// TIA Portal V17 export
// export: Created 2022-07-28T18:02:48.2971435Z, ExportSetting None, DisplayName Totally Integrated Automation Portal, DisplayVersion V17, DisplayName TIA Portal Openness, DisplayVersion V17, DisplayName TIA Portal Teamcenter Gateway, DisplayVersion V17, DisplayName TIA Portal Version Control Interface, DisplayVersion V17, DisplayName TIA Portal Test Suite Advanced, DisplayVersion V17, DisplayName SINAMICS Startdrive Advanced, DisplayVersion V17, DisplayName SINAMICS DCC, DisplayVersion V17, DisplayName SINAMICS Startdrive G130, G150, S120, S150, SINAMICS MV, S210, DisplayVersion V17, DisplayName SINAMICS Startdrive G110M, G120, G120C, G120D, G120P, G115D, DisplayVersion V17, DisplayName STEP 7 Professional, DisplayVersion V17, DisplayName SIMATIC Energy Suite, DisplayVersion V17, DisplayName STEP 7 CFC, DisplayVersion V17, DisplayName STEP 7 Safety, DisplayVersion V17, DisplayName WinCC Advanced / Unified PC, DisplayVersion V17, DisplayName SIMATIC Visualization Architect, DisplayVersion V17
FUNCTION "PID_FC" : Void   // FC21, SCL
{ S7_Optimized_Access := 'TRUE' }
// stored: AutoNumber false, SetENOAutomatically false
   VAR_TEMP
      t_SupplyRelease : Bool;   // 1 - Release from supply
   END_VAR
BEGIN
   #t_SupplyRelease := true;

   REGION (ID = 18) Регулятор температути вихідної води 1 TIC_W1011
       //Тип елемента: ПІД

       REGION Блокування та зовнішні аварії
           REGION Блокування Open
               "D_TIC_W1011_Ctrl".IB_InterlocksOpen_8.%X0 := false;
               "D_TIC_W1011_Ctrl".IB_InterlocksOpen_8.%X1 := false;
               "D_TIC_W1011_Ctrl".IB_InterlocksOpen_8.%X2 := false;
               "D_TIC_W1011_Ctrl".IB_InterlocksOpen_8.%X3 := false;
               "D_TIC_W1011_Ctrl".IB_InterlocksOpen_8.%X4 := false;
               "D_TIC_W1011_Ctrl".IB_InterlocksOpen_8.%X5 := false;
               "D_TIC_W1011_Ctrl".IB_InterlocksOpen_8.%X6 := false;
               "D_TIC_W1011_Ctrl".IB_InterlocksOpen_8.%X7 := false;
           END_REGION

           REGION Блокування Close
               "D_TIC_W1011_Ctrl".IB_InterlocksClose_8.%X0 := false;
               "D_TIC_W1011_Ctrl".IB_InterlocksClose_8.%X1 := false;
               "D_TIC_W1011_Ctrl".IB_InterlocksClose_8.%X2 := false;
               "D_TIC_W1011_Ctrl".IB_InterlocksClose_8.%X3 := false;
               "D_TIC_W1011_Ctrl".IB_InterlocksClose_8.%X4 := false;
               "D_TIC_W1011_Ctrl".IB_InterlocksClose_8.%X5 := false;
               "D_TIC_W1011_Ctrl".IB_InterlocksClose_8.%X6 := false;
               "D_TIC_W1011_Ctrl".IB_InterlocksClose_8.%X7 := false;
           END_REGION

           REGION Зовнішні аварії та попередження
               "D_TIC_W1011_Ctrl".IW_ExternalError_16.%X0 := false;
               "D_TIC_W1011_Ctrl".IW_ExternalError_16.%X1 := false;
               "D_TIC_W1011_Ctrl".IW_ExternalError_16.%X2 := false;
               "D_TIC_W1011_Ctrl".IW_ExternalError_16.%X3 := false;
               "D_TIC_W1011_Ctrl".IW_ExternalError_16.%X4 := false;
               "D_TIC_W1011_Ctrl".IW_ExternalError_16.%X5 := false;
               "D_TIC_W1011_Ctrl".IW_ExternalError_16.%X6 := false;
               "D_TIC_W1011_Ctrl".IW_ExternalError_16.%X7 := false;
               "D_TIC_W1011_Ctrl".IW_ExternalError_16.%X8 := false;
               "D_TIC_W1011_Ctrl".IW_ExternalError_16.%X9 := false;
               "D_TIC_W1011_Ctrl".IW_ExternalError_16.%X10 := false;
               "D_TIC_W1011_Ctrl".IW_ExternalError_16.%X11 := false;
               "D_TIC_W1011_Ctrl".IW_ExternalError_16.%X12 := false;
               "D_TIC_W1011_Ctrl".IW_ExternalError_16.%X13 := false;
               "D_TIC_W1011_Ctrl".IW_ExternalError_16.%X14 := false;
               "D_TIC_W1011_Ctrl".IW_ExternalError_16.%X15 := false;

               "D_N1Gr_Ctrl".I_ExternalWarning := false;
           END_REGION
       END_REGION

       REGION Блок керування



           "D_TIC_W1011_Ctrl"(I_Initialization := "D_General_ProgramDATA".RestartPLC,
                              IR_CycleTime := "D_PLC".TIME_TCK.cyclic_sec_R,
                              II_Obj_ID := 18,
                              I_CmdGeneralReset := "D_General_ProgramDATA".ResetGlobal,
                              I_One_1s := "D_PLC".PLS.P1S,
                              I_EstopHMI := "D_General_ProgramDATA".ES_HMI_Global
                              AND "D_General_ProgramDATA".ES_Fld_Global,
                              IR_MinOut := 35.0,
                              IR_MaxOut := 100.0,
                              IR_CyclePID := 0.1,
                              II_ID_Sensor := 4,
                              QI_Out_PID => "D_InOut"."TIC_W1011".QI_AnalogValue,
                              IQ_PLC_CycleInfo := "D_PLC_CycleInfo_DATA".Grp_Obj[1, 0]);
       END_REGION

   END_REGION

   REGION (ID = 19) Регулятор температути вихідної води 2 TIC_811
       //Тип елемента: ПІД

       REGION Блокування та зовнішні аварії
           REGION Блокування Open
               "D_TIC_811_Ctrl".IB_InterlocksOpen_8.%X0 := false;
               "D_TIC_811_Ctrl".IB_InterlocksOpen_8.%X1 := false;
               "D_TIC_811_Ctrl".IB_InterlocksOpen_8.%X2 := false;
               "D_TIC_811_Ctrl".IB_InterlocksOpen_8.%X3 := false;
               "D_TIC_811_Ctrl".IB_InterlocksOpen_8.%X4 := false;
               "D_TIC_811_Ctrl".IB_InterlocksOpen_8.%X5 := false;
               "D_TIC_811_Ctrl".IB_InterlocksOpen_8.%X6 := false;
               "D_TIC_811_Ctrl".IB_InterlocksOpen_8.%X7 := false;
           END_REGION

           REGION Блокування Close
               "D_TIC_811_Ctrl".IB_InterlocksClose_8.%X0 := false;
               "D_TIC_811_Ctrl".IB_InterlocksClose_8.%X1 := false;
               "D_TIC_811_Ctrl".IB_InterlocksClose_8.%X2 := false;
               "D_TIC_811_Ctrl".IB_InterlocksClose_8.%X3 := false;
               "D_TIC_811_Ctrl".IB_InterlocksClose_8.%X4 := false;
               "D_TIC_811_Ctrl".IB_InterlocksClose_8.%X5 := false;
               "D_TIC_811_Ctrl".IB_InterlocksClose_8.%X6 := false;
               "D_TIC_811_Ctrl".IB_InterlocksClose_8.%X7 := false;
           END_REGION

           REGION Зовнішні аварії та попередження
               "D_TIC_811_Ctrl".IW_ExternalError_16.%X0 := false;
               "D_TIC_811_Ctrl".IW_ExternalError_16.%X1 := false;
               "D_TIC_811_Ctrl".IW_ExternalError_16.%X2 := false;
               "D_TIC_811_Ctrl".IW_ExternalError_16.%X3 := false;
               "D_TIC_811_Ctrl".IW_ExternalError_16.%X4 := false;
               "D_TIC_811_Ctrl".IW_ExternalError_16.%X5 := false;
               "D_TIC_811_Ctrl".IW_ExternalError_16.%X6 := false;
               "D_TIC_811_Ctrl".IW_ExternalError_16.%X7 := false;
               "D_TIC_811_Ctrl".IW_ExternalError_16.%X8 := false;
               "D_TIC_811_Ctrl".IW_ExternalError_16.%X9 := false;
               "D_TIC_811_Ctrl".IW_ExternalError_16.%X10 := false;
               "D_TIC_811_Ctrl".IW_ExternalError_16.%X11 := false;
               "D_TIC_811_Ctrl".IW_ExternalError_16.%X12 := false;
               "D_TIC_811_Ctrl".IW_ExternalError_16.%X13 := false;
               "D_TIC_811_Ctrl".IW_ExternalError_16.%X14 := false;
               "D_TIC_811_Ctrl".IW_ExternalError_16.%X15 := false;

               "D_N1Gr_Ctrl".I_ExternalWarning := false;
           END_REGION
       END_REGION

       REGION Блок керування



           "D_TIC_811_Ctrl"(I_Initialization := "D_General_ProgramDATA".RestartPLC,
                            IR_CycleTime := "D_PLC".TIME_TCK.cyclic_sec_R,
                            II_Obj_ID := 19,
                            I_CmdGeneralReset := "D_General_ProgramDATA".ResetGlobal,
                            I_One_1s := "D_PLC".PLS.P1S,
                            I_EstopHMI := "D_General_ProgramDATA".ES_HMI_Global
                            AND "D_General_ProgramDATA".ES_Fld_Global,
                            IR_MinOut := 25.0,
                            IR_MaxOut := 100.0,
                            IR_CyclePID := 0.1,
                            II_ID_Sensor := 5,
                            QI_Out_PID => "D_InOut"."TIC_811".QI_AnalogValue,
                            IQ_PLC_CycleInfo := "D_PLC_CycleInfo_DATA".Grp_Obj[1, 0]);
       END_REGION

   END_REGION

   REGION (ID = 20) Регулятор тиску кислоти LIC_PW579CA
       //Тип елемента: ПІД

       REGION Блокування та зовнішні аварії
           REGION Блокування Open
               "D_LIC_PW579CA_Ctrl".IB_InterlocksOpen_8.%X0 := false;
               "D_LIC_PW579CA_Ctrl".IB_InterlocksOpen_8.%X1 := false;
               "D_LIC_PW579CA_Ctrl".IB_InterlocksOpen_8.%X2 := false;
               "D_LIC_PW579CA_Ctrl".IB_InterlocksOpen_8.%X3 := false;
               "D_LIC_PW579CA_Ctrl".IB_InterlocksOpen_8.%X4 := false;
               "D_LIC_PW579CA_Ctrl".IB_InterlocksOpen_8.%X5 := false;
               "D_LIC_PW579CA_Ctrl".IB_InterlocksOpen_8.%X6 := false;
               "D_LIC_PW579CA_Ctrl".IB_InterlocksOpen_8.%X7 := false;
           END_REGION

           REGION Блокування Close
               "D_LIC_PW579CA_Ctrl".IB_InterlocksClose_8.%X0 := false;
               "D_LIC_PW579CA_Ctrl".IB_InterlocksClose_8.%X1 := false;
               "D_LIC_PW579CA_Ctrl".IB_InterlocksClose_8.%X2 := false;
               "D_LIC_PW579CA_Ctrl".IB_InterlocksClose_8.%X3 := false;
               "D_LIC_PW579CA_Ctrl".IB_InterlocksClose_8.%X4 := false;
               "D_LIC_PW579CA_Ctrl".IB_InterlocksClose_8.%X5 := false;
               "D_LIC_PW579CA_Ctrl".IB_InterlocksClose_8.%X6 := false;
               "D_LIC_PW579CA_Ctrl".IB_InterlocksClose_8.%X7 := false;
           END_REGION

           REGION Зовнішні аварії та попередження
               "D_LIC_PW579CA_Ctrl".IW_ExternalError_16.%X0 := false;
               "D_LIC_PW579CA_Ctrl".IW_ExternalError_16.%X1 := false;
               "D_LIC_PW579CA_Ctrl".IW_ExternalError_16.%X2 := false;
               "D_LIC_PW579CA_Ctrl".IW_ExternalError_16.%X3 := false;
               "D_LIC_PW579CA_Ctrl".IW_ExternalError_16.%X4 := false;
               "D_LIC_PW579CA_Ctrl".IW_ExternalError_16.%X5 := false;
               "D_LIC_PW579CA_Ctrl".IW_ExternalError_16.%X6 := false;
               "D_LIC_PW579CA_Ctrl".IW_ExternalError_16.%X7 := false;
               "D_LIC_PW579CA_Ctrl".IW_ExternalError_16.%X8 := false;
               "D_LIC_PW579CA_Ctrl".IW_ExternalError_16.%X9 := false;
               "D_LIC_PW579CA_Ctrl".IW_ExternalError_16.%X10 := false;
               "D_LIC_PW579CA_Ctrl".IW_ExternalError_16.%X11 := false;
               "D_LIC_PW579CA_Ctrl".IW_ExternalError_16.%X12 := false;
               "D_LIC_PW579CA_Ctrl".IW_ExternalError_16.%X13 := false;
               "D_LIC_PW579CA_Ctrl".IW_ExternalError_16.%X14 := false;
               "D_LIC_PW579CA_Ctrl".IW_ExternalError_16.%X15 := false;

               "D_N1Gr_Ctrl".I_ExternalWarning := false;
           END_REGION
       END_REGION

       REGION Блок керування



           "D_LIC_PW579CA_Ctrl"(I_Initialization := "D_General_ProgramDATA".RestartPLC,
                                IR_CycleTime := "D_PLC".TIME_TCK.cyclic_sec_R,
                                II_Obj_ID := 20,
                                I_CmdGeneralReset := "D_General_ProgramDATA".ResetGlobal,
                                I_One_1s := "D_PLC".PLS.P1S,
                                I_EstopHMI := "D_General_ProgramDATA".ES_HMI_Global
                                AND "D_General_ProgramDATA".ES_Fld_Global,
                                IR_MinOut := 25.0,
                                IR_MaxOut := 100.0,
                                IR_CyclePID := 0.1,
                                II_ID_Sensor := 30,
                                QI_Out_PID => "D_InOut"."LIC_PW579CA".QI_AnalogValue,
                                IQ_PLC_CycleInfo := "D_PLC_CycleInfo_DATA".Grp_Obj[1, 0]);
       END_REGION

   END_REGION

   REGION (ID = 21) Регулятор тиску лугу LIC_PW579NA
       //Тип елемента: ПІД

       REGION Блокування та зовнішні аварії
           REGION Блокування Open
               "D_LIC_PW579NA_Ctrl".IB_InterlocksOpen_8.%X0 := false;
               "D_LIC_PW579NA_Ctrl".IB_InterlocksOpen_8.%X1 := false;
               "D_LIC_PW579NA_Ctrl".IB_InterlocksOpen_8.%X2 := false;
               "D_LIC_PW579NA_Ctrl".IB_InterlocksOpen_8.%X3 := false;
               "D_LIC_PW579NA_Ctrl".IB_InterlocksOpen_8.%X4 := false;
               "D_LIC_PW579NA_Ctrl".IB_InterlocksOpen_8.%X5 := false;
               "D_LIC_PW579NA_Ctrl".IB_InterlocksOpen_8.%X6 := false;
               "D_LIC_PW579NA_Ctrl".IB_InterlocksOpen_8.%X7 := false;
           END_REGION

           REGION Блокування Close
               "D_LIC_PW579NA_Ctrl".IB_InterlocksClose_8.%X0 := false;
               "D_LIC_PW579NA_Ctrl".IB_InterlocksClose_8.%X1 := false;
               "D_LIC_PW579NA_Ctrl".IB_InterlocksClose_8.%X2 := false;
               "D_LIC_PW579NA_Ctrl".IB_InterlocksClose_8.%X3 := false;
               "D_LIC_PW579NA_Ctrl".IB_InterlocksClose_8.%X4 := false;
               "D_LIC_PW579NA_Ctrl".IB_InterlocksClose_8.%X5 := false;
               "D_LIC_PW579NA_Ctrl".IB_InterlocksClose_8.%X6 := false;
               "D_LIC_PW579NA_Ctrl".IB_InterlocksClose_8.%X7 := false;
           END_REGION

           REGION Зовнішні аварії та попередження
               "D_LIC_PW579NA_Ctrl".IW_ExternalError_16.%X0 := false;
               "D_LIC_PW579NA_Ctrl".IW_ExternalError_16.%X1 := false;
               "D_LIC_PW579NA_Ctrl".IW_ExternalError_16.%X2 := false;
               "D_LIC_PW579NA_Ctrl".IW_ExternalError_16.%X3 := false;
               "D_LIC_PW579NA_Ctrl".IW_ExternalError_16.%X4 := false;
               "D_LIC_PW579NA_Ctrl".IW_ExternalError_16.%X5 := false;
               "D_LIC_PW579NA_Ctrl".IW_ExternalError_16.%X6 := false;
               "D_LIC_PW579NA_Ctrl".IW_ExternalError_16.%X7 := false;
               "D_LIC_PW579NA_Ctrl".IW_ExternalError_16.%X8 := false;
               "D_LIC_PW579NA_Ctrl".IW_ExternalError_16.%X9 := false;
               "D_LIC_PW579NA_Ctrl".IW_ExternalError_16.%X10 := false;
               "D_LIC_PW579NA_Ctrl".IW_ExternalError_16.%X11 := false;
               "D_LIC_PW579NA_Ctrl".IW_ExternalError_16.%X12 := false;
               "D_LIC_PW579NA_Ctrl".IW_ExternalError_16.%X13 := false;
               "D_LIC_PW579NA_Ctrl".IW_ExternalError_16.%X14 := false;
               "D_LIC_PW579NA_Ctrl".IW_ExternalError_16.%X15 := false;

               "D_N1Gr_Ctrl".I_ExternalWarning := false;
           END_REGION
       END_REGION

       REGION Блок керування



           "D_LIC_PW579NA_Ctrl"(I_Initialization := "D_General_ProgramDATA".RestartPLC,
                                IR_CycleTime := "D_PLC".TIME_TCK.cyclic_sec_R,
                                II_Obj_ID := 21,
                                I_CmdGeneralReset := "D_General_ProgramDATA".ResetGlobal,
                                I_One_1s := "D_PLC".PLS.P1S,
                                I_EstopHMI := "D_General_ProgramDATA".ES_HMI_Global
                                AND "D_General_ProgramDATA".ES_Fld_Global,
                                IR_MinOut := 25.0,
                                IR_MaxOut := 100.0,
                                IR_CyclePID := 0.1,
                                II_ID_Sensor := 31,
                                QI_Out_PID => "D_InOut"."LIC_PW579NA".QI_AnalogValue,
                                IQ_PLC_CycleInfo := "D_PLC_CycleInfo_DATA".Grp_Obj[1, 0]);
       END_REGION

   END_REGION

   REGION (ID = 22) Регулятор тиску технологічної води PIC_PW0_W
       //Тип елемента: ПІД

       REGION Блокування та зовнішні аварії
           REGION Блокування Open
               "D_PIC_PW0_W_Ctrl".IB_InterlocksOpen_8.%X0 := false;
               "D_PIC_PW0_W_Ctrl".IB_InterlocksOpen_8.%X1 := false;
               "D_PIC_PW0_W_Ctrl".IB_InterlocksOpen_8.%X2 := false;
               "D_PIC_PW0_W_Ctrl".IB_InterlocksOpen_8.%X3 := false;
               "D_PIC_PW0_W_Ctrl".IB_InterlocksOpen_8.%X4 := false;
               "D_PIC_PW0_W_Ctrl".IB_InterlocksOpen_8.%X5 := false;
               "D_PIC_PW0_W_Ctrl".IB_InterlocksOpen_8.%X6 := false;
               "D_PIC_PW0_W_Ctrl".IB_InterlocksOpen_8.%X7 := false;
           END_REGION

           REGION Блокування Close
               "D_PIC_PW0_W_Ctrl".IB_InterlocksClose_8.%X0 := false;
               "D_PIC_PW0_W_Ctrl".IB_InterlocksClose_8.%X1 := false;
               "D_PIC_PW0_W_Ctrl".IB_InterlocksClose_8.%X2 := false;
               "D_PIC_PW0_W_Ctrl".IB_InterlocksClose_8.%X3 := false;
               "D_PIC_PW0_W_Ctrl".IB_InterlocksClose_8.%X4 := false;
               "D_PIC_PW0_W_Ctrl".IB_InterlocksClose_8.%X5 := false;
               "D_PIC_PW0_W_Ctrl".IB_InterlocksClose_8.%X6 := false;
               "D_PIC_PW0_W_Ctrl".IB_InterlocksClose_8.%X7 := false;
           END_REGION

           REGION Зовнішні аварії та попередження
               "D_PIC_PW0_W_Ctrl".IW_ExternalError_16.%X0 := false;
               "D_PIC_PW0_W_Ctrl".IW_ExternalError_16.%X1 := false;
               "D_PIC_PW0_W_Ctrl".IW_ExternalError_16.%X2 := false;
               "D_PIC_PW0_W_Ctrl".IW_ExternalError_16.%X3 := false;
               "D_PIC_PW0_W_Ctrl".IW_ExternalError_16.%X4 := false;
               "D_PIC_PW0_W_Ctrl".IW_ExternalError_16.%X5 := false;
               "D_PIC_PW0_W_Ctrl".IW_ExternalError_16.%X6 := false;
               "D_PIC_PW0_W_Ctrl".IW_ExternalError_16.%X7 := false;
               "D_PIC_PW0_W_Ctrl".IW_ExternalError_16.%X8 := false;
               "D_PIC_PW0_W_Ctrl".IW_ExternalError_16.%X9 := false;
               "D_PIC_PW0_W_Ctrl".IW_ExternalError_16.%X10 := false;
               "D_PIC_PW0_W_Ctrl".IW_ExternalError_16.%X11 := false;
               "D_PIC_PW0_W_Ctrl".IW_ExternalError_16.%X12 := false;
               "D_PIC_PW0_W_Ctrl".IW_ExternalError_16.%X13 := false;
               "D_PIC_PW0_W_Ctrl".IW_ExternalError_16.%X14 := false;
               "D_PIC_PW0_W_Ctrl".IW_ExternalError_16.%X15 := false;

               "D_N1Gr_Ctrl".I_ExternalWarning := false;
           END_REGION
       END_REGION

       REGION Блок керування



           "D_PIC_PW0_W_Ctrl"(I_Initialization := "D_General_ProgramDATA".RestartPLC,
                              IR_CycleTime := "D_PLC".TIME_TCK.cyclic_sec_R,
                              II_Obj_ID := 22,
                              I_CmdGeneralReset := "D_General_ProgramDATA".ResetGlobal,
                              I_One_1s := "D_PLC".PLS.P1S,
                              I_EstopHMI := "D_General_ProgramDATA".ES_HMI_Global
                              AND "D_General_ProgramDATA".ES_Fld_Global,
                              IR_MinOut := 25.0,
                              IR_MaxOut := 100.0,
                              IR_CyclePID := 0.1,
                              II_ID_Sensor := 35,
                              QI_Out_PID => "D_InOut"."PIC_PW0_W".QI_AnalogValue,
                              IQ_PLC_CycleInfo := "D_PLC_CycleInfo_DATA".Grp_Obj[1, 0]);
       END_REGION

   END_REGION

   REGION (ID = 23) Регулятор тиску оборотної води PIC_N_Gr
       //Тип елемента: ПІД каскадний

       REGION Блокування та зовнішні аварії
           REGION Блокування Open
               "D_PIC_N_Gr_Ctrl".IB_InterlocksOpen_8.%X0 := false;
               "D_PIC_N_Gr_Ctrl".IB_InterlocksOpen_8.%X1 := false;
               "D_PIC_N_Gr_Ctrl".IB_InterlocksOpen_8.%X2 := false;
               "D_PIC_N_Gr_Ctrl".IB_InterlocksOpen_8.%X3 := false;
               "D_PIC_N_Gr_Ctrl".IB_InterlocksOpen_8.%X4 := false;
               "D_PIC_N_Gr_Ctrl".IB_InterlocksOpen_8.%X5 := false;
               "D_PIC_N_Gr_Ctrl".IB_InterlocksOpen_8.%X6 := false;
               "D_PIC_N_Gr_Ctrl".IB_InterlocksOpen_8.%X7 := false;
           END_REGION

           REGION Блокування Close
               "D_PIC_N_Gr_Ctrl".IB_InterlocksClose_8.%X0 := false;
               "D_PIC_N_Gr_Ctrl".IB_InterlocksClose_8.%X1 := false;
               "D_PIC_N_Gr_Ctrl".IB_InterlocksClose_8.%X2 := false;
               "D_PIC_N_Gr_Ctrl".IB_InterlocksClose_8.%X3 := false;
               "D_PIC_N_Gr_Ctrl".IB_InterlocksClose_8.%X4 := false;
               "D_PIC_N_Gr_Ctrl".IB_InterlocksClose_8.%X5 := false;
               "D_PIC_N_Gr_Ctrl".IB_InterlocksClose_8.%X6 := false;
               "D_PIC_N_Gr_Ctrl".IB_InterlocksClose_8.%X7 := false;
           END_REGION

           REGION Зовнішні аварії та попередження
               "D_PIC_N_Gr_Ctrl".IW_ExternalError_16.%X0 := false;
               "D_PIC_N_Gr_Ctrl".IW_ExternalError_16.%X1 := false;
               "D_PIC_N_Gr_Ctrl".IW_ExternalError_16.%X2 := false;
               "D_PIC_N_Gr_Ctrl".IW_ExternalError_16.%X3 := false;
               "D_PIC_N_Gr_Ctrl".IW_ExternalError_16.%X4 := false;
               "D_PIC_N_Gr_Ctrl".IW_ExternalError_16.%X5 := false;
               "D_PIC_N_Gr_Ctrl".IW_ExternalError_16.%X6 := false;
               "D_PIC_N_Gr_Ctrl".IW_ExternalError_16.%X7 := false;
               "D_PIC_N_Gr_Ctrl".IW_ExternalError_16.%X8 := false;
               "D_PIC_N_Gr_Ctrl".IW_ExternalError_16.%X9 := false;
               "D_PIC_N_Gr_Ctrl".IW_ExternalError_16.%X10 := false;
               "D_PIC_N_Gr_Ctrl".IW_ExternalError_16.%X11 := false;
               "D_PIC_N_Gr_Ctrl".IW_ExternalError_16.%X12 := false;
               "D_PIC_N_Gr_Ctrl".IW_ExternalError_16.%X13 := false;
               "D_PIC_N_Gr_Ctrl".IW_ExternalError_16.%X14 := false;
               "D_PIC_N_Gr_Ctrl".IW_ExternalError_16.%X15 := false;

               "D_N1Gr_Ctrl".I_ExternalWarning := false;
           END_REGION
       END_REGION

       REGION Блок керування

           "D_PIC_N_Gr_Ctrl".IA_ID_Inv[0] := 14;
           "D_PIC_N_Gr_Ctrl".IA_ID_Inv[1] := 15;
           "D_PIC_N_Gr_Ctrl".IA_ID_Inv[2] := 16;

           "D_PIC_N_Gr_Ctrl"(I_Initialization := "D_General_ProgramDATA".RestartPLC,
                             IR_CycleTime := "D_PLC".TIME_TCK.cyclic_sec_R,
                             II_Obj_ID := 23,
                             I_CmdGeneralReset := "D_General_ProgramDATA".ResetGlobal,
                             I_One_1s := "D_PLC".PLS.P1S,
                             I_EstopHMI := "D_General_ProgramDATA".ES_HMI_Global
                             AND "D_General_ProgramDATA".ES_Fld_Global,
                             IR_MinOut := 25.0,
                             IR_MaxOut := 100.0,
                             IR_CyclePID := 0.1,
                             II_ID_Sensor := 3,
                             II_Num_Inv := 3,
                             IQ_PLC_CycleInfo := "D_PLC_CycleInfo_DATA".Grp_Obj[1, 0]);
       END_REGION

   END_REGION
END_FUNCTION
